// TwinCAT 3 PLC project LCLSVacuum
// Title: LCLSVacuumLib
// Company: SLAC
// Author: Alex Wallace & Scott Stubbs
// ProjectVersion: 1.12.6969
// Description: No serial drivers exist in this library. Need LCLSVacuumSerialDrivers for that. 1.2.0 ecat diagnostic 1.2.1 added the ecat lib in here 1.2.2 adding the ratio check function for valve interlocking 1.3.6 added 275 & 500 gauges, minor changes 1.4.0 added a normally open gate valve structure and FB 1.5.0 added error and warning codes to ptm structure for pfeiffers 1.5.1 seamless override open/close on vgc during transition from override to normal mode. 1.7.0 ST_PTM now uses inheritence model. Started implementing Ebara support. 1.8.0 Moved to seperate functions for 937A and 937B controllers.
// ProgramVersion: 3.1.4023.0
// libraries:
//   LCLS General,0.1.2,SLAC
//   Tc2_EtherCAT, * (Beckhoff Automation GmbH)
//   Tc2_Standard, * (Beckhoff Automation GmbH)
//   Tc2_System, * (Beckhoff Automation GmbH)
//   Tc2_TcpIp, * (Beckhoff Automation GmbH)
//   Tc2_Utilities, * (Beckhoff Automation GmbH)
//   Tc3_Interfaces, * (Beckhoff Automation GmbH)
//   Tc3_Module, * (Beckhoff Automation GmbH)
// project tree:
//   Data types/Gauges/ E_PressureState.TcDUT (not stored), Gauge_Type.TcDUT (not stored), ST_VG.TcDUT (not stored)
//   Data types/IO/ IO_EP2338.TcDUT (not stored)
//   Data types/ ISG_Struct.TcDUT (not stored), ST_Encoder.TcDUT (not stored), UpStrInVac_Struct.TcDUT (not stored), UpStrOutVac_Struct.TcDUT (not stored)
//   Data types/Pumps/ E_PumpState.TcDUT (not stored), ST_AgilentControlStatus.TcDUT (not stored), ST_AgilentPTM.TcDUT (not stored), ST_AuxiliaryPump.TcDUT (not stored), ST_EbaraDryPump.TcDUT (not stored), ST_EbaraPTM.TcDUT (not stored), ST_LeyboldPTM.TcDUT (not stored), ST_PfeifferPTM.TcDUT (not stored), ST_PIP.TcDUT (not stored), ST_PTM.TcDUT (not stored), ST_ReadbackOnlyPump.TcDUT (not stored), ST_RoughPump.TcDUT (not stored)
//   Data types/Valves/ E_VCN.TcDUT (not stored), E_ValvePositionState.TcDUT (not stored), E_VGC.TcDUT (not stored), ST_VCC.TcDUT (not stored), ST_VCC_NO.TcDUT (not stored), ST_VCN.TcDUT (not stored), ST_VGC.TcDUT (not stored), ST_VGC_NO.TcDUT (not stored), ST_VRC.TcDUT (not stored)
//   Global Variables/ Constants.TcGVL (not stored), Global_Variables.TcGVL (not stored)
//   POUs/ Example_GaugeSup.TcPOU (not stored)
//   POUs/Functions/Gauge FB/ FB_500.TcPOU (not stored), FB_903.TcPOU (not stored), FB_907.TcPOU (not stored), FB_275.TcPOU (not stored), FB_909.TcPOU (not stored), FB_925.TcPOU, FB_937A_VG.TcPOU (not stored), FB_937B_VG.TcPOU (not stored), FB_972.TcPOU (not stored), FB_Dumb_Gauge.TcPOU (not stored), FB_PressureState.TcPOU (not stored), FB_GCM.TcPOU (not stored), FB_GGO.TcPOU
//   POUs/Functions/Pumps/ FB_EbaraDryPump.TcPOU (not stored), FB_PTM_Pfeiffer.TcPOU (not stored), FB_PTM_Ebara.TcPOU (not stored), FB_PTM_Agilent.TcPOU (not stored), FB_PTM_MagDriveDigital.TcPOU (not stored), FB_PTM_LeyboldTD20Classic.TcPOU (not stored), FB_ScrollPump.TcPOU (not stored), FB_TurboExtLogic.TcPOU (not stored), FB_VARIAN301TURBO.TcPOU (not stored)
//   POUs/Functions/Valve FB/ FB_TurbVentvalve_NO.TcPOU (not stored), FB_VCC_NO.TcPOU (not stored), FB_VCN.TcPOU (not stored), FB_VGC.TcPOU (not stored), FB_VGC_NO.TcPOU (not stored), FB_VRC.TcPOU (not stored), FB_VCC.TcPOU (not stored), FB_VRC_OK_CLS.TcPOU (not stored), F_VALVE_REL_ILK.TcPOU (not stored), F_VRC_DIODE_ILK.TcPOU (not stored), F_TURBO_VRC_ILK.TcPOU (not stored)
//   Version/ Global_Version.TcGVL

// ---- Version/Global_Version.TcGVL
{attribute 'TcGenerated'}
{attribute 'no-analysis'}
{attribute 'linkalways'}
// This function has been automatically generated from the project information.
VAR_GLOBAL CONSTANT
	{attribute 'const_non_replaced'}
	stLibVersion_LCLSVacuumLib : ST_LibVersion := (iMajor := 1, iMinor := 12, iBuild := 6969, iRevision := 0, sVersion := '1.12.6969');
END_VAR

// ---- POUs/Functions/Gauge FB/FB_925.TcPOU
FUNCTION_BLOCK FB_925
VAR_INPUT
END_VAR
VAR_OUTPUT
END_VAR
VAR_IN_OUT
	VG	: ST_VG;
END_VAR
VAR
	rV : REAL;
	fbGaugeState : FB_PressureState;
	rMaxPressure	:	REAL := 760; //Torr
	rMinPressure	:	REAL := 1E-5; //Torr
END_VAR

(* Standard MKS 9XX series conversion *)
(* works for 972 and 925 *)

//Default setpoint 50 mT
IF VG.rVAC_SP = 0 THEN
	VG.rVAC_SP := 5E-2;
END_IF

rV := 10*INT_TO_REAL(VG.iPRESS_R)/32767;

IF rV >= 0.99 THEN
	IF rV >= 0.99 AND rV < 1 THEN
		VG.rPRESS := 1E-5;
	ELSE
		VG.rPRESS := LREAL_TO_REAL(EXPT(10, REAL_TO_LREAL(rV-6)));
	END_IF
	VG.xPRESS_OK := TRUE; //Backwards compatibility
ELSE
	VG.xPRESS_OK := FALSE;
END_IF

(* Pressure OK check *)
fbGaugeState.i_rV := rV;
fbGaugeState.i_MaxPressure := rMaxPressure;
fbGaugeState.i_MinPressure := rMinPressure;
fbGaugeState(iq_stVG:=VG);

(* Setpoint evaluation *)
VG.xAT_VAC := VG.xPRESS_OK AND (VG.rPRESS < VG.rVAC_SP);

END_FUNCTION_BLOCK

// ---- POUs/Functions/Gauge FB/FB_GGO.TcPOU
FUNCTION_BLOCK FB_GGO
VAR_IN_OUT
	iq_astGauges: ARRAY[0..gc_iSizeOfGGOArray] OF ST_VG;
	iq_axHV_RO: ARRAY[0..gc_iSizeOfGGOArray] OF BOOL;
END_VAR
VAR_INPUT
	i_iIndex: INT;
END_VAR
VAR

	stPG: ST_VG;
	stVG: ST_VG;
	//index for associated pirani
	wPG : WORD;

	
	// FBs
	fb903	:	FB_903;
	fb907	:	FB_907;
	fb909	:	FB_909;
	fb925	:	FB_925;
	fbGCM	:	FB_GCM;
	
END_VAR

(* This function block is used to calculate the pressure from the analog input voltage and to provide protection and automatic turn on of ion gauges.
 It also manages the turn on fo the AT_VAC boolean, and checks to make sure the pressure is good *)

(* Full-scale pressure conversion factor *)

(* Real-value voltage calculation *)
(* Generic expression for pressure in the MKS systems

P = 10^(V/0.6-12)

722B = 0
903 = 1
907 = 2
909 = 3
925 = 4

*)

(* Make a copy of gauge at index*)
stVG := iq_astGauges[LIMIT(0 ,i_iIndex, gc_iSizeOfGGOArray)];

(* Check that it is an ion gauge *)
IF stVG.eTYPE = Gauge_Type.IG903 OR stVG.eTYPE = Gauge_Type.IG909 THEN

(* Check that Associated Gauge is within index*)
	IF WORD_TO_INT(stVG.wPG) <= gc_iSizeOfGGOArray THEN
		(* Check pressure gauge type before assignment *)
		(* Add high pressure gauge types here *)
		IF iq_astGauges[stVG.wPG].eTYPE = PG722B OR //722B
		iq_astGauges[stVG.wPG].eTYPE = PG907 OR //907
		iq_astGauges[stVG.wPG].eTYPE = PG925 THEN //925
			stPG := iq_astGauges[stVG.wPG];  (* Copy associated pirani gauge number to local variable *)
		ELSE //Default to allow the IG to turn on, this allows someone to set the PG to another IG and turn the gauge on whenever they want
			stPG.rPRESS := 1E-3;
			stPG.xPRESS_OK := TRUE;
		END_IF
	
	END_IF
END_IF

(* Evaluate each Gauge pressure based on eTYPE*)
CASE iq_astGauges[i_iIndex].eTYPE OF
	
	//Baratron Gauge
	PG722B:
		fbGCM(VG:=iq_astGauges[i_iIndex]);
		
	//Cold Cathode
	Gauge_Type.IG903:
		fb903(IG:=iq_astGauges[i_iIndex], PG:=iq_astGauges[wPG]);
		
	//Pirani Gauge	
	PG907:
		fb907(PG:=iq_astGauges[i_iIndex]);
		
	//Hot Cathode	
	Gauge_Type.IG909:
		fb909(IG:=iq_astGauges[i_iIndex], PG:=iq_astGauges[wPG]);
		
	//MicroPirani Gauge	
	PG925:
		fb925(VG:=iq_astGauges[i_iIndex]);
	ELSE
		(* Now, since we don't know what gauge type we're dealing with, we want 
		to make sure to reset all the gauge parameters, otherwise we may be 
		left with stale information *)
	stVG.rPRESS := 760;
	stVG.xAT_VAC := FALSE;
	stVG.xPRESS_OK := FALSE;
	stVG.xHV_SW := FALSE;
		
END_CASE

(* reAssign "HV On" back into High Voltage Array*)
iq_axHV_RO[LIMIT(0,WORD_TO_INT(stVG.wHV_RO),gc_iSizeOfGGOArray)]:=stVG.xHV_DIS;

END_FUNCTION_BLOCK
